{attribute 'qualified_only'}
{attribute 'strict'}
TYPE ST_MCK_ParIn :
STRUCT
	rTareSetting			:REAL;//皮重设置
	rTarePresetValue		:REAL;//预置皮重设定
	
END_STRUCT
END_TYPE

(* stored: Version 1.1.0.1, ProductVersion 3.1.4024.9
   DUT ST_MCK_ParIn: Id {6e7cbec0-483b-495c-8ac3-d1c232537824} *)
